FUNCTION_BLOCK PointerTaskExample
VAR
	_parameter : I_ParameterPosition;
	_status	   : POINTER TO ParameterSet;
END_VAR

METHOD CyclicLogic
VAR_INPUT
END_VAR
IF _parameter = 0 OR _status = 0 THEN
	RETURN;
END_IF
_status^.Position := _parameter.Position;
END_METHOD

//FB_Init is always available implicitly and it is used primarily for initialization.
//The return value is not evaluated. For a specific influence, you can also declare the
//methods explicitly and provide additional code there with the standard initialization
//code. You can evaluate the return value.
METHOD FB_Init: BOOL
VAR_INPUT
    bInitRetains: BOOL; // TRUE: the retain variables are initialized (reset warm / reset cold)
    bInCopyCode: BOOL;  // TRUE: the instance will be copied to the copy code afterward (online change)   
	Mover : I_Mover;
END_VAR
_parameter := Mover.Parameters;
__QUERYPOINTER(Mover.Status,_Status);
END_METHOD

END_FUNCTION_BLOCK

(* stored: Version 1.1.0.1
   POU PointerTaskExample: Id {13908b64-3e2b-4c4c-a38f-3c72e669e0b8}, SpecialFunc None
   Method CyclicLogic: Id {eb4da503-4e6e-49f9-8c6d-b38b2ef47199}
   Method FB_Init: Id {37956a57-2694-4fad-ad90-f5f58c7a227e} *)
